{attribute 'qualified_only'}
{attribute 'strict'}
TYPE KlantToestand :
(
	voorBalie := 0,
	wordtGeholpen,
	aanHetWachten,
	heeftVerf
);
END_TYPE

(* stored: Version 1.1.0.1, ProductVersion 3.1.4024.15
   DUT KlantToestand: Id {55f94cf3-191f-43b4-aa73-bae45694b309} *)
